(* LS Electric XG5000 project: Nitra_FB *)
(* PLC LSPLC *)
(* module base 0 slot 0: Input/Output Module:XEM-DN/DP32HP (DC 24V Input, Transistor Output, 32 Contacts) *)
(* module base 0 slot 1: Internal Positioning:XBF-PO06E (Open Collector Type, 6 Axis) *)
(* module base 0 slot 2: EtherNet/IP:XBL-EIPT (EtherNet/IP communication module, electrical) *)
VAR_GLOBAL
    Pal_EIP_Input00 : ARRAY[0..145] OF BYTE; (* Input data to ethernet/IP Nitra PAL-EIP *)
    Pal_EIP_Output00 : ARRAY[0..101] OF BYTE; (* Output data to ethernet/IP Nitra PAL-EIP *)
    Pal_EIP_Unit00 : PAL_EIP_UDT;
END_VAR

(* Comments on direct variables
%IX0.0.0	this is comment 1
*)

TYPE PAL_EIP_UDT : (* Data type for accessing inputs and outputs of a Nitra PAL EIP manifold. *)
STRUCT
    DigitalInput_08pt_Module : ARRAY[0..15] OF BYTE; (* Input data from 8 point digital input modules. *)
    DigitalInput_16pt_Module : ARRAY[0..7] OF WORD; (* Input data from 16 point digital input modules. *)
    AnalogInput_RawData : ARRAY[0..15] OF INT; (* Analog input data unscaled. *)
    TemperatureInput_ImpliedDecimal : ARRAY[0..15] OF INT; (* Temperature module inputs *)
    DigitalOutput_06pt_Module : ARRAY[0..21] OF BYTE; (* Digital output data for 6 point modules. *)
    DigitalOutput_08pt_Module : ARRAY[0..15] OF BYTE; (* Digital output data for 8 point modules. *)
    DigitalOutput_16pt_Module : ARRAY[0..7] OF WORD; (* Digital output data for 16 point modules. *)
    AnalogOutput_RawData : ARRAY[0..15] OF INT; (* Analog output data unscaled *)
    DiagnosticData : USINT; (* Nitra Pal diagnostic data *)
    Valve : ARRAY[0..127] OF BOOL; (* Control Pneumatic valves connected to PAL unit *)
END_STRUCT;
END_TYPE

FUNCTION_BLOCK Nitra_PAL_MapData_FB
VAR_INPUT
    Enable : BOOL; (* Enable the FB. *)
    Source_InputData : ARRAY[0..145] OF BYTE; (* This is the input data from EIP Block of Nitra PAL in the P2P settings. *)
END_VAR
VAR_IN_OUT
    Source_OutputData : ARRAY[0..101] OF BYTE; (* This is the output data from EIP Block of Nitra PAL in the P2P settings. *)
    PAL_User_UDT : PAL_EIP_UDT; (* This is the user data type created for this PAL manifold. *)
END_VAR
VAR_OUTPUT
    Active : BOOL; (* status that function block is enabled. *)
END_VAR
VAR
    boolCount00 : INT; (* array count variable for looping. *)
    boolCount01 : INT; (* array count variable for looping. *)
    boolCount02 : INT; (* array count variable for looping. *)
    boolCount03 : INT; (* array count variable for looping. *)
    boolCount04 : INT; (* array count variable for looping. *)
    boolCount05 : INT; (* array count variable for looping. *)
    boolCount06 : INT; (* array count variable for looping. *)
    boolCount07 : INT; (* array count variable for looping. *)
    byteCount : INT; (* array counting variable *)
    byteCount2 : INT; (* array counting variable *)
    Destination_OutputData : ARRAY[0..101] OF BYTE; (* Data to be copied into Source_OutputData after every loop. *)
    i : INT; (* array variable *)
    Temporary_BYTE : ARRAY[0..63] OF BYTE; (* Temporary storage of byte data *)
    Temporary_BYTE2 : BYTE; (* temporary byte storage *)
    Temporary_BYTE3 : BYTE; (* temporary byte storage. *)
    Temporary_WORD : WORD; (* temporary word storage. *)
END_VAR
(* 
AutomationDirect.com has provided this code for convenience. This sample code is provided "as-is" with no expressed or implied warranty. 
 If the end user includes any of the sample code (in whole or part), it is the user's responsibility to completely modify, integrate, and test any code to ensure it meets all system and 
 safety requirements for the intended application or system.
 *)

(* Only run function block if enable is true *)
IF (Enable = TRUE) THEN
		Active := TRUE;
	
		(************************************************************
         		Copy Diagnostic Data
   		************************************************************ *)
		PAL_User_UDT.DiagnosticData := BYTE_TO_USINT(IN:=Source_InputData[0]);
		
		
		
		(************************************************************
         		Copy 8 pt Digital Inputs
   		************************************************************ *)
		PAL_User_UDT.DigitalInput_08pt_Module :=  ARY_MOVE(MOVE_NUM:=16, IN:=Source_InputData, IN_INDX:=1, OUT_INDX:=0);
		
		
		(************************************************************
         		Copy 16 pt Digital Inputs
   		************************************************************ *)
		(* Loop through 16 pt digital input to put it in to temporary byte storage*)	
		byteCount := 97;
		byteCount2 := byteCount + 1;
		
		FOR i:=0 TO 7 BY 1 DO
			
			Temporary_BYTE2 := Source_InputData[byteCount];
			Temporary_BYTE3 := Source_InputData[byteCount2];
			
			Temporary_WORD :=BYTE_WORD(LOW:=Temporary_BYTE2, HIGH:=Temporary_BYTE3);
			
	 		PAL_User_UDT.DigitalInput_16pt_Module[i] := Temporary_WORD;
			
			byteCount := byteCount + 2;
			byteCount2 := byteCount + 1;
		
		END_FOR;
		
		
		(************************************************************
         		Copy Analog Inputs
   		************************************************************ *)	
		(* Loop through analog input data to put it in to temporary byte storage*)	
		byteCount := 17;
		byteCount2 := byteCount + 1;
		
		FOR i:=0 TO 15 BY 1 DO
			
			Temporary_BYTE2 := Source_InputData[byteCount];
			Temporary_BYTE3 := Source_InputData[byteCount2];
			
			Temporary_WORD :=BYTE_WORD(LOW:=Temporary_BYTE2, HIGH:=Temporary_BYTE3);
			
	 		PAL_User_UDT.AnalogInput_RawData[i] :=WORD_TO_INT(IN:=Temporary_WORD);
			
			byteCount := byteCount + 2;
			byteCount2 := byteCount + 1;
		
		END_FOR;
		
		
		(************************************************************
         		Copy Temperature Inputs
   		************************************************************ *)	
		(* Loop through temperature input data to put it in to temporary byte storage*)	
		byteCount := 113;
		byteCount2 := byteCount + 1;
		
		FOR i:=0 TO 15 BY 1 DO
			
			Temporary_BYTE2 := Source_InputData[byteCount];
			Temporary_BYTE3 := Source_InputData[byteCount2];
			
			Temporary_WORD :=BYTE_WORD(LOW:=Temporary_BYTE2, HIGH:=Temporary_BYTE3);
			
	 		PAL_User_UDT.TemperatureInput_ImpliedDecimal[i] :=WORD_TO_INT(IN:=Temporary_WORD);
			
			byteCount := byteCount + 2;
			byteCount2 := byteCount + 1;
		
		END_FOR;
			
			
			
			
			
			
			
			
			
		(************************************************************
         		Copy Valve Outputs 
   		************************************************************ *)
		boolCount00 := 0;
		boolCount01 := boolCount00 + 1;
		boolCount02 := boolCount01 + 1;
		boolCount03 := boolCount02 + 1;
		boolCount04 := boolCount03 + 1;
		boolCount05 := boolCount04 + 1;
		boolCount06 := boolCount05 + 1;
		boolCount07 := boolCount06 + 1;
		
		(* Loop through temporary byte array to pack valve booleans in to it. *)	
		FOR i:=0 TO 63 BY 1 DO
			
			
			Temporary_BYTE[i] := BIT_BYTE(EN:= TRUE, IN1:=PAL_User_UDT.Valve[boolCount00], IN2:=PAL_User_UDT.Valve[boolCount01], IN3:=PAL_User_UDT.Valve[boolCount02], IN4:=PAL_User_UDT.Valve[boolCount03], IN5:=PAL_User_UDT.Valve[boolCount04], IN6:=PAL_User_UDT.Valve[boolCount05], IN7:=PAL_User_UDT.Valve[boolCount06], IN8:=PAL_User_UDT.Valve[boolCount07]);
			
						
			boolCount00 := boolCount00 + 8;
			boolCount01 := boolCount00 + 1;
			boolCount02 := boolCount01 + 1;
			boolCount03 := boolCount02 + 1;
			boolCount04 := boolCount03 + 1;
			boolCount05 := boolCount04 + 1;
			boolCount06 := boolCount05 + 1;
			boolCount07 := boolCount06 + 1;
		
		END_FOR;
		
		(* Copy valve output byte packing to temporary output array *)	
		Destination_OutputData :=  ARY_MOVE(MOVE_NUM:=64, IN:=Temporary_BYTE, IN_INDX:=0, OUT_INDX:=0);
			
			
		(************************************************************
	 		Copy 6 point output data to temporary output array 
		***************************************************************)
		Destination_OutputData :=  ARY_MOVE(MOVE_NUM:=22, IN:=PAL_User_UDT.DigitalOutput_06pt_Module, IN_INDX:=0, OUT_INDX:=32);
		
		(************************************************************
	 		Copy 8 point output data to temporary output array 
		***************************************************************)
		Destination_OutputData :=  ARY_MOVE(MOVE_NUM:=16, IN:=PAL_User_UDT.DigitalOutput_08pt_Module, IN_INDX:=0, OUT_INDX:=16);
		
		(************************************************************
	 		Copy 16 point output data to temporary output array 
		***************************************************************)
		
		
		(* Loop through 16 point digital output data to put it in to temporary byte storage*)	
		byteCount := 0;
		byteCount2 := byteCount + 1;
		
		FOR i:=0 TO 15 BY 1 DO
			
			WORD_BYTE(IN:=PAL_User_UDT.DigitalOutput_16pt_Module[i], LOW=>Temporary_BYTE[byteCount], HIGH=>Temporary_BYTE[byteCount2]);
			
			byteCount := i + 2;
			byteCount2 := byteCount + 1;
		
		END_FOR;
		
		Destination_OutputData :=  ARY_MOVE(MOVE_NUM:=16, IN:=Temporary_BYTE, IN_INDX:=0, OUT_INDX:=86);
		
		
		(************************************************************
	 		Copy analog output data to temporary output array 
		***************************************************************)
		(* Loop through analog output data to put it in to temporary byte storage*)	
		byteCount := 0;
		byteCount2 := byteCount + 1;
		
		FOR i:=0 TO 15 BY 1 DO
			Temporary_WORD :=INT_TO_WORD(IN:=PAL_User_UDT.AnalogOutput_RawData[i]);
			WORD_BYTE(IN:=Temporary_WORD, LOW=>Temporary_BYTE[byteCount], HIGH=>Temporary_BYTE[byteCount2]);
			
			byteCount := byteCount + 2;
			byteCount2 := byteCount + 1;
		
		END_FOR;
		
		Destination_OutputData :=  ARY_MOVE(MOVE_NUM:=32, IN:=Temporary_BYTE, IN_INDX:=0, OUT_INDX:=54);
	
	
		(* Copy temporary output data array to the source output that gets sent to the PAL unit *)
		Source_OutputData := ARY_MOVE(MOVE_NUM:= 102, IN:=Destination_OutputData, IN_INDX:=0, OUT_INDX:=0);

ELSE	
	Active := FALSE;
	
END_IF; //end of enable if
END_FUNCTION_BLOCK

PROGRAM FB_Usage_LD (* task: Scan Program *)
VAR
    Pal_EIP_00 : Nitra_PAL_MapData_FB;
END_VAR
VAR_EXTERNAL
    Pal_EIP_Input00 : ARRAY[0..145] OF BYTE; (* Input data to ethernet/IP Nitra PAL-EIP *)
    Pal_EIP_Output00 : ARRAY[0..101] OF BYTE; (* Output data to ethernet/IP Nitra PAL-EIP *)
    Pal_EIP_Unit00 : PAL_EIP_UDT;
END_VAR

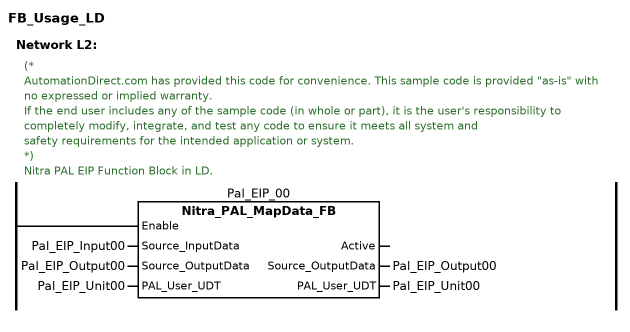
(* ( * / AutomationDirect.com has provided this code for convenience. This sample code is provided "as-is" with no expressed or implied warranty. / If the end user includes any of the sample code (in whole or part), it is the user's responsibility to completely modify, integrate, and test any code to ensure it meets all system and / safety requirements for the intended application or system. / * ) *)
(* Nitra PAL EIP Function Block in LD. *)
(* Rung L2 *)
Pal_EIP_00(Enable := TRUE, Source_InputData := Pal_EIP_Input00, Source_OutputData := Pal_EIP_Output00, PAL_User_UDT := Pal_EIP_Unit00, Source_OutputData => Pal_EIP_Output00, PAL_User_UDT => Pal_EIP_Unit00);
END_PROGRAM

PROGRAM FB_Usage_ST (* task: Scan Program *)
(*  *)
VAR
    fbActive : BOOL;
    Pal_EIP_00 : Nitra_PAL_MapData_FB;
END_VAR
VAR_EXTERNAL
    Pal_EIP_Input00 : ARRAY[0..145] OF BYTE; (* Input data to ethernet/IP Nitra PAL-EIP *)
    Pal_EIP_Output00 : ARRAY[0..101] OF BYTE; (* Output data to ethernet/IP Nitra PAL-EIP *)
    Pal_EIP_Unit00 : PAL_EIP_UDT;
END_VAR
(* 
AutomationDirect.com has provided this code for convenience. This sample code is provided "as-is" with no expressed or implied warranty. 
 If the end user includes any of the sample code (in whole or part), it is the user's responsibility to completely modify, integrate, and test any code to ensure it meets all system and 
 safety requirements for the intended application or system.
 *)
Pal_EIP_00(Enable:=TRUE, Source_InputData:=Pal_EIP_Input00, Source_OutputData:=Pal_EIP_Output00, PAL_User_UDT:=Pal_EIP_Unit00, Active=>fbActive);
END_PROGRAM